// Mitsubishi GX Works2 project: 스캔2 램프하나씩 키기   PLC: Q02/Q02H

PROGRAM MAIN
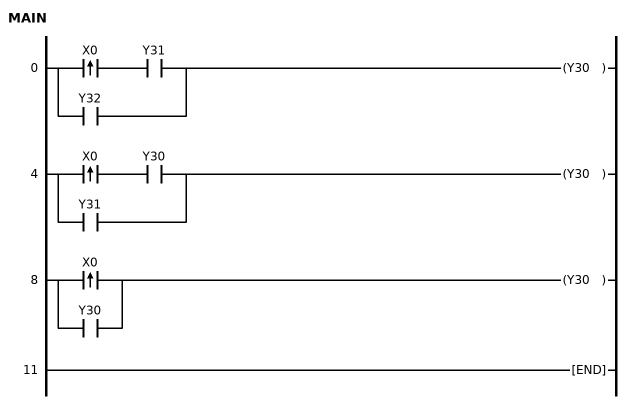
0     LDP     X0
      AND     Y31
      OR      Y32
      OUT     Y30
4     LDP     X0
      AND     Y30
      OR      Y31
      OUT     Y30
8     LDP     X0
      OR      Y30
      OUT     Y30
11    END
END_PROGRAM
